// TwinCAT 3 PLC project CBox
// ProgramVersion: 3.1.4023.0
// libraries:
//   Tc2_Standard, * (Beckhoff Automation GmbH)
//   Tc2_System, * (Beckhoff Automation GmbH)
//   Tc3_Module, * (Beckhoff Automation GmbH)
// project tree:
//   / GlobalTextList.TcGTLO, PlcTask.TcTTO, Visualization Manager.TcVMO (not stored)
//   InputControlBox/ InputGVL_ControlBox.TcGVL, ST_RealBoxParams.TcDUT
//   POUs/ MAIN.TcPOU
//   VirtualControlBox/FBs + Methods/ FB_CtrlBox.TcPOU, FC_ReadJoyPos.TcPOU
//   VirtualControlBox/ GVL_ControlBox.TcGVL, HMI_ControlBox.TcVIS, ST_BoxParams.TcDUT
//   VirtualControlBox/Interfaces/ ITF_ControlBox.TcIO
// real-time tasks:
//   TASK PlcTask: cycle T#10ms, priority 20, ADS port 350

CONFIGURATION CBox
    RESOURCE PLC ON TwinCAT3
        TASK PlcTask(INTERVAL := T#10ms, PRIORITY := 20);
        PROGRAM MAIN WITH PlcTask : MAIN;
    END_RESOURCE
END_CONFIGURATION

// ---- InputControlBox/ST_RealBoxParams.TcDUT
TYPE ST_RealBoxParams :
STRUCT
	Start : BOOL;
	Stop : BOOL;
	Off : BOOL;
	Auto : BOOL;
	Manual : BOOL;
	TopSwitch : BOOL;
	JOY_X : REAL;
	JOY_Y : REAL; 
END_STRUCT
END_TYPE

// ---- VirtualControlBox/ST_BoxParams.TcDUT
TYPE ST_BoxParams :
STRUCT
	Start : BOOL;
	Stop : BOOL;
	Off : BOOL;
	Auto : BOOL;
	Manual : BOOL;
	TopSwitch : BOOL;
	JOY_X : REAL;
	JOY_Y : REAL; 
END_STRUCT
END_TYPE

// ---- InputControlBox/InputGVL_ControlBox.TcGVL
{attribute 'qualified_only'}
VAR_GLOBAL
	stRealControlParams : ST_RealBoxParams; 
END_VAR

// ---- VirtualControlBox/GVL_ControlBox.TcGVL
{attribute 'qualified_only'}
VAR_GLOBAL
	stControlParams : ST_BoxParams; 
END_VAR

// ---- VirtualControlBox/Interfaces/ITF_ControlBox.TcIO
INTERFACE ITF_ControlBox EXTENDS FB_CtrlBox

END_INTERFACE

// ---- POUs/MAIN.TcPOU
PROGRAM MAIN
VAR
	bmanSelect : BOOL := ST_BoxParams.Manual; 
	bAutoSelect : BOOL := ST_BoxParams.Auto; 
	bStart : BOOL := ST_BoxParams.Start;
	bStop : BOOL := ST_BoxParams.Stop; 
END_VAR

END_PROGRAM

// ---- VirtualControlBox/FBs + Methods/FB_CtrlBox.TcPOU
FUNCTION_BLOCK FB_CtrlBox
VAR_INPUT
END_VAR
VAR_OUTPUT
END_VAR
VAR
	
END_VAR

METHOD CheckStatus : BOOL
VAR_INPUT
	bOff : BOOL;
	bAuto : BOOL;
	bManual : BOOL; 
	bStartButton : BOOL;
	bStopButton : BOOL; 
	fClockSignal : REAL; 
	fPipePressure : REAL;
	bSensorError : BOOL; 
END_VAR
VAR_OUTPUT
	bNotReady : BOOL; 
	bReady : BOOL; 
	bStarting : BOOL;
	bRunning : BOOL; 
	bStopping : BOOL; 
	bError : BOOL; 
	bGreenLight : BOOL;
	bRedLight : BOOL; 
	dCurrentStatus : INT; 
	
END_VAR
IF bOff AND NOT bManual AND NOT bAuto THEN
	bNotReady := TRUE; 
	dCurrentStatus := 1;
	
ELSIF bManual OR bAuto THEN
	bReady := TRUE; 
	dCurrentStatus := 2;
	
ELSIF bStartButton AND NOT bRunning THEN
	bStarting := TRUE; 
	dCurrentStatus := 3;
	
ELSIF (bManual AND bStartButton) OR (bAuto AND bStartButton AND fClockSignal > 0) THEN
	bRunning := TRUE; 
	bGreenLight := TRUE; 
	dCurrentStatus := 4;
	
ELSIF (bStopButton AND bRunning) THEN
	bStopping := TRUE;
	bRedLight := TRUE; 
	dCurrentStatus := 5;
	
ELSIF (fPipePressure < 10 OR bSensorError := TRUE) THEN
	bError := TRUE; 
	bRedLight := TRUE; 
	dCurrentStatus := 6; 
END_IF
END_METHOD

METHOD JoyStick : REAL
VAR_INPUT
	dMachineStatus : INT; 
	bTopSwitch : BOOL; 
	bManMode : BOOL; 
	dBoxSelect : INT; 
	dJoyStickWinch : INT;
	dJoyStickCyl : INT; 
END_VAR
VAR_OUTPUT
	fJoyStickPosX : REAL;  
	fJoyStickPosY : REAL; 
END_VAR
VAR
	ControlBox : REFERENCE TO GVL_ControlBox; 
END_VAR


IF (bManMode = TRUE) AND (dMachineStatus = 4) AND bTopSwitch = TRUE THEN
	IF dBoxSelect = 1 THEN
		ControlBox := GVL_ControlBox;
		fJoyStickPosX := GVL_ControlBox.stControlParams.JOY_X; 
		fJoyStickPosY := GVL_ControlBox.stControlParams.JOY_Y; 
	ELSE
		ControlBox := InputGVL_ControlBox;
		fJoyStickPosX := InputGVL_ControlBox.stRealControlParams.JOY_X/32767;
		fJoyStickPosY := InputGVL_ControlBox.stRealControlParams.JOY_Y/32767;  	
			
	END_IF
	
	
	
END_IF
END_METHOD

METHOD ModeSelection : BOOL
VAR_INPUT
	bInOff : BOOL;
	bInAuto : BOOL;
	bInManual : BOOL; 
END_VAR
VAR_OUTPUT
	bOutOff : BOOL;
	bOutAuto : BOOL;
	bOutManual : BOOL; 
END_VAR

IF NOT bInOff AND NOT bInAuto THEN
	bOutManual := TRUE;
ELSIF NOT bInOff AND NOT bInManual THEN
	bOutAuto := TRUE; 
ELSE
	bInOff := TRUE;
END_IF
END_METHOD

END_FUNCTION_BLOCK

// ---- VirtualControlBox/FBs + Methods/FC_ReadJoyPos.TcPOU
FUNCTION FC_ReadJoyPos : REAL
VAR_INPUT
END_VAR
VAR
END_VAR

END_FUNCTION

// ---- GlobalTextList.TcGTLO
TEXTLIST GlobalTextList
  30 = 'AUTO'
  68 = 'AUTO ON'
  829 = 'AutoModeOn'
  604 = 'CylinderControl'
  6 = 'MANUAL'
  758 = 'ManualModeOn'
  310 = 'OFF'
  845 = 'Start'
  442 = 'START'
  32 = 'STOP'
  740 = "STOP'"
  518 = 'WinchControl'
END_TEXTLIST

// ---- VirtualControlBox/HMI_ControlBox.TcVIS
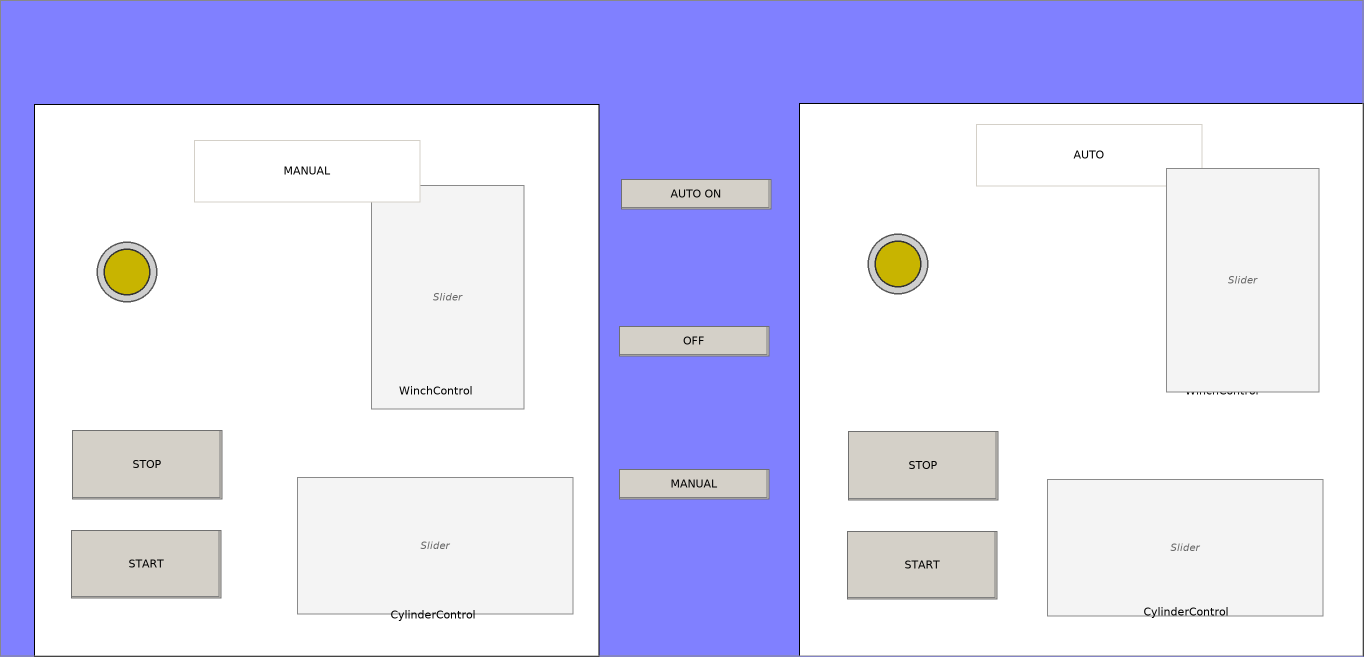
VISUALIZATION HMI_ControlBox  // 1364x657
    Rectangle (34,104 565x553)
    Button (71,530 150x68), "START"
        tap GVL_ControlBox.stControlParams.Start
    Button (72,430 150x69), "STOP"
        tap GVL_ControlBox.stControlParams.Stop
    Slider (297,477 276x137), variable: GVL_ControlBox.stControlParams.JOY_X, scale -1..1
    Slider (371,185 153x224), variable: GVL_ControlBox.stControlParams.JOY_Y, scale 1..-1
    Textfield (194,140 226x62), "MANUAL", input disabled if: GVL_ControlBox.stControlParams.Auto
    Rectangle (799,103 565x553)
    Textfield (976,124 226x62), "AUTO", input disabled if: GVL_ControlBox.stControlParams.Manual
    Button (847,531 150x68), "START"
        tap GVL_ControlBox.stControlParams.Start
    Button (848,431 150x69), "STOP"
        tap GVL_ControlBox.stControlParams.Stop
    Slider (1047,479 276x137), variable: GVL_ControlBox.stControlParams.JOY_X, scale -1..1
    Lamp1 (92,237 70x70), tooltip "ManualModeOn", variable: GVL_ControlBox.stControlParams.Manual, style: Lamp-Lamp1-Yellow
    Lamp1 (863,229 70x70), tooltip "AutoModeOn", variable: GVL_ControlBox.stControlParams.Auto, style: Lamp-Lamp1-Yellow
    Button (621,179 150x30), "AUTO ON"
    Button (619,326 150x30), "OFF"
    Button (619,469 150x30), "MANUAL"
    Label (1111,597 150x30), "CylinderControl"
    Label (358,600 150x30), "CylinderControl"
    Label (361,376 150x30), "WinchControl"
    Label (1147,376 150x30), "WinchControl"
    Slider (1166,168 153x224), variable: GVL_ControlBox.stControlParams.JOY_Y, scale 1..-1
END_VISUALIZATION
